# EPICS StreamDevice protocol: picoIOC/protocols/NewFocus8742.proto
OutTerminator = CR;
InTerminator = CR LF;

getIPAddress{
	out "IPADDR?";
	in "%s";
}

move_relative{
	out "%(\$1)iPR%i";
}

getVelo{
	out "%(\$1)iVA?";
	in "%i";
}

setVelo{
	out "%(\$1)iVA%i";
}

getPos{
	out "%(\$1)iPA?";
	in "%i";
}
